// Mitsubishi GX Works2 project: FrekvensM   PLC: FX1S

// global labels: Global1
VAR_GLOBAL
  Giv_1 AT X001 : BOOL;  (* Givare 1 *)
  Giv_2 AT X002 : BOOL;  (* Givare 2 *)
  Giv_3 AT X003 : BOOL;  (* Givare 3 *)
  Giv_4 AT X004 : BOOL;  (* Givare 4 *)
  FR AT Y000 : BOOL;  (* Start FRAM *)
  BK AT Y001 : BOOL;  (* Start BACK *)
  MD AT Y002 : BOOL;  (* Hastighet Medium *)
  LO AT Y003 : BOOL;  (* Hastighet Låg *)
  HI AT Y004 : BOOL;  (* Hastighet Hög *)
END_VAR

// task Task_01 (event TRUE, interval 0, priority 31): POU_01

PROGRAM POU_01
(* 3 olika hastigheter ut PÅ/AV (HI, MD, LO)
	PÅ/AV FRAM (FR)
	PÅ/AV BACK (BK)*)
	
(* START KNAPP in, 
	4 givare in Giv1, Giv2, Giv3, Giv4 (simuleras med knappar) *)
	
(* Intern start-signal START för att underlätta repetition. *)

(* Sätt frekvensomvandlare acc/dec till 3Hz/sek *)
	
WHILE START = TRUE DO
	IF Giv1 = TRUE THEN
		FR = TRUE AND LO = TRUE
	END_IF;	
END_WHILE;
END_PROGRAM
